(* CoDeSys 2.3.9.52 project: test.pro *)
(* Libraries: Standard.lib 20.5.14 09:13:26, Iecsfc.lib 30.1.13 14:05:12, SYSLIBCALLBACK.LIB 30.1.13 14:05:12 *)

(* POU PLC_PRG, ST *)
PROGRAM PLC_PRG
VAR
	a:BOOL;
	b:REAL;
	c:STRING;
	TON:TON;
END_VAR
TON(IN:=NOT(TON.Q), PT:=T#200ms);
IF TON.Q THEN
	IF b>100 THEN b:=0; END_IF;
	b:=b+1;
END_IF;
END_PROGRAM

(* POU Configuration/MODBUS_CONFIGURATION, ST *)
PROGRAM MODBUS_CONFIGURATION        
VAR                                
END_VAR                            
(*                                 
   <?xml version="1.0" encoding="UTF-16" standalone="yes"?>
<network xml_structure_version="1" xml_feature_version="1">
	<generator_settings minRTUTaskCycleTimeMs="5" minEthaskCycleTimeMs="5" ethSlaveMultiplier="0.1" rtuInterfaceMultiplier="0.1" taskGeneration="true"/>
</network>
                              
*)                                 
;                                  
END_PROGRAM
